FUNCTION_BLOCK CompRegister
VAR_GENERIC CONSTANT
	nCap	: UDINT := 100;
END_VAR

IMPLEMENTS I_MutCompRegister

VAR
	_iRegister	: ARRAY[1..nCap] OF I_Component;
	_nLen		: UDINT := 0;
END_VAR

PROPERTY Cap : UDINT
GET
Cap := nCap;
END_GET
END_PROPERTY

METHOD Get : Result
VAR_INPUT
	nIndex		: UDINT;
END_VAR
VAR_OUTPUT
	iComp	: I_Component;
END_VAR
IF _nLen = 0 THEN
	RETURN;
END_IF

IF nIndex > _nLen THEN
	RETURN;
END_IF

IF nIndex > nCap OR_ELSE nIndex < 1 THEN
	Get := Err.Ovf;
	RETURN;
END_IF

iComp := _iRegister[nIndex];
Get := Ok;
END_METHOD

METHOD Insert : Result
VAR_INPUT
	iComponent	: I_Component;
END_VAR
VAR_OUTPUT
	nIndex		: UDINT;
END_VAR
VAR
	i			: UDINT;
END_VAR
IF iComponent = 0 THEN
	Insert := Err.Itf0;
	RETURN;
END_IF

IF _nLen = nCap THEN
	Insert := Err.Ovf;
	RETURN;
END_IF

FOR i := 1 TO _nLen DO
	IF _iRegister[i] = iComponent THEN		
		Insert := Err.ItfEq;
		RETURN;	
	END_IF
END_FOR

_nLen := _nLen + 1;
_iRegister[_nLen] := iComponent;
Insert := Ok;
END_METHOD

PROPERTY Length : UDINT
GET
Length := _nLen;
END_GET
END_PROPERTY

END_FUNCTION_BLOCK

(* stored: Version 1.1.0.1
   POU CompRegister: Id {ca518f37-6c05-4cf4-89d4-75c5e2201c82}, SpecialFunc None
   Property Cap: Id {50df78aa-587a-44e1-afbf-df9af1ffc7cc}
   Get Get: Id {dfda453b-d7cf-4f39-afd5-c17fcce041a4}
   Method Get: Id {54d36c41-e48b-4d94-a7f2-51e33876950d}
   Method Insert: Id {9fb06efd-ab03-4fa1-aa5f-6a55026b07b7}
   Property Length: Id {6bac9759-9382-43e1-accb-7021bbfc1551}
   Get Get: Id {464d3f9b-7d83-4738-a4f1-48441410ea69} *)
